SUBAPPLICATION QueryServiceHTTPSub (* Query services using HTTP with the service defined *)
  (* Standard: 61499-2; Description: Copyright (c) 2019 fortiss GmbH This program and the accompanying materials are made available under the terms of the Eclipse Public License 2.0 which is available at https://www.eclipse.org/legal/epl-2.0/ SPDX-License-Identifier: PL-2.0 *)
  (* Version 1.0, 2019-02-05, Jose Cabral, fortiss GmbH *)
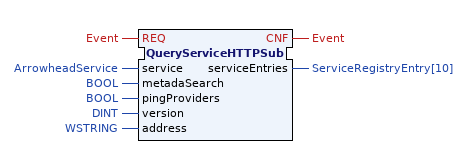
  EVENT_INPUT
    REQ; (* Query for services *)
  END_EVENT
  EVENT_OUTPUT
    CNF; (* Query finished *)
  END_EVENT
  VAR_INPUT
    service : ArrowheadService; (* The Arrowhead Service object that is looked for (SD and supported IDD-s) *)
    metadaSearch : BOOL; (* True, if service metadata shall be taken into account during query *)
    pingProviders : BOOL; (* True, if the selected (query fitting) Application Systems shall be pinged to see if they’re alive *)
    version : DINT; (* The minimum version of the Service we are looking for *)
    address : WSTRING; (* Address of the Service Registry (not officially in the documentation, but it simplifies the FBs) *)
  END_VAR
  VAR_OUTPUT
    serviceEntries : ARRAY [0..9] OF ServiceRegistryEntry;
  END_VAR
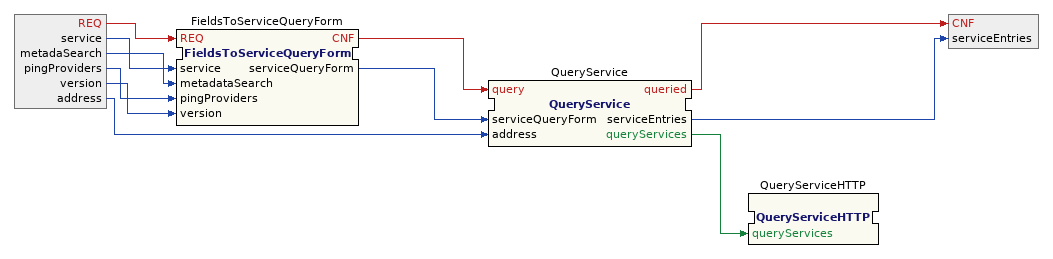
  FBS
    FieldsToServiceQueryForm : FieldsToServiceQueryForm;
    QueryService : QueryService;
    QueryServiceHTTP : QueryServiceHTTP;
  END_FBS
  EVENT_CONNECTIONS
    FieldsToServiceQueryForm.CNF TO QueryService.query;
    QueryService.queried TO CNF;
    REQ TO FieldsToServiceQueryForm.REQ;
  END_CONNECTIONS
  DATA_CONNECTIONS
    FieldsToServiceQueryForm.serviceQueryForm TO QueryService.serviceQueryForm;
    QueryService.serviceEntries TO serviceEntries;
    service TO FieldsToServiceQueryForm.service;
    metadaSearch TO FieldsToServiceQueryForm.metadataSearch;
    pingProviders TO FieldsToServiceQueryForm.pingProviders;
    version TO FieldsToServiceQueryForm.version;
    address TO QueryService.address;
  END_CONNECTIONS
  ADAPTER_CONNECTIONS
    QueryService.queryServices TO QueryServiceHTTP.queryServices;
  END_CONNECTIONS
END_SUBAPPLICATION
